// Mitsubishi GX Works2 project: plc0807   PLC: Q03UDV

PROGRAM MAIN
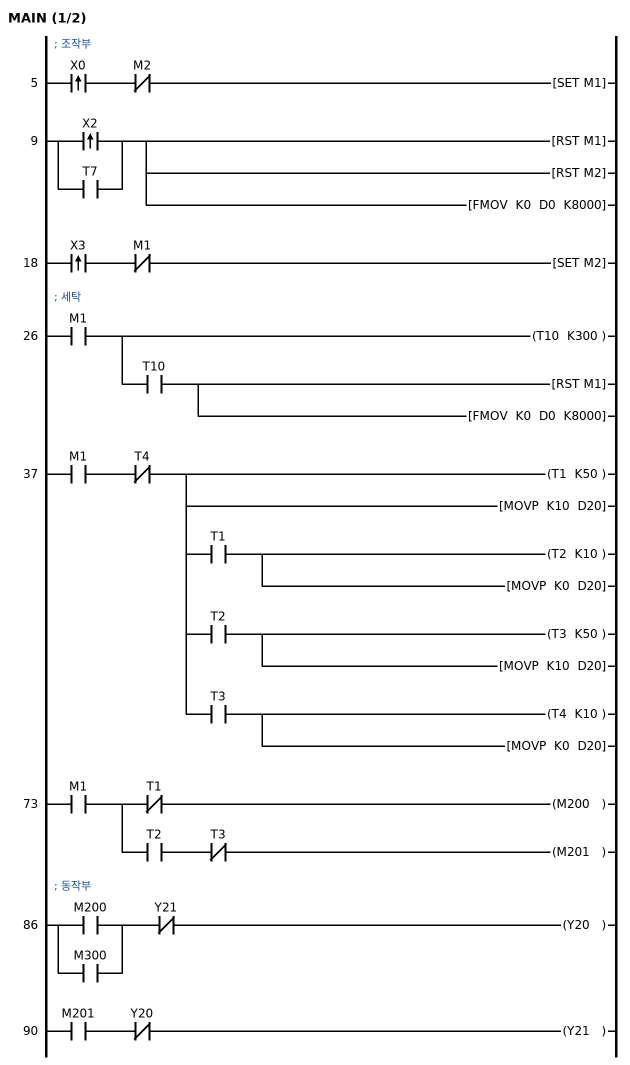
; 조작부
5     LDP     X0
      ANI     M2
      SET     M1
9     LDP     X2
      OR      T7
      RST     M1
      RST     M2
      FMOV    K0 D0 K8000
18    LDP     X3
      ANI     M1
      SET     M2
; 세탁
26    LD      M1
      OUT     T10 K300
      AND     T10
      RST     M1
      FMOV    K0 D0 K8000
37    LD      M1
      ANI     T4
      OUT     T1 K50
      MOVP    K10 D20
      MPS
      AND     T1
      OUT     T2 K10
      MOVP    K0 D20
      MRD
      AND     T2
      OUT     T3 K50
      MOVP    K10 D20
      MPP
      AND     T3
      OUT     T4 K10
      MOVP    K0 D20
73    LD      M1
      MPS
      ANI     T1
      OUT     M200
      MPP
      AND     T2
      ANI     T3
      OUT     M201
; 동작부
86    LD      M200
      OR      M300
      ANI     Y21
      OUT     Y20
90    LD      M201
      ANI     Y20
      OUT     Y21
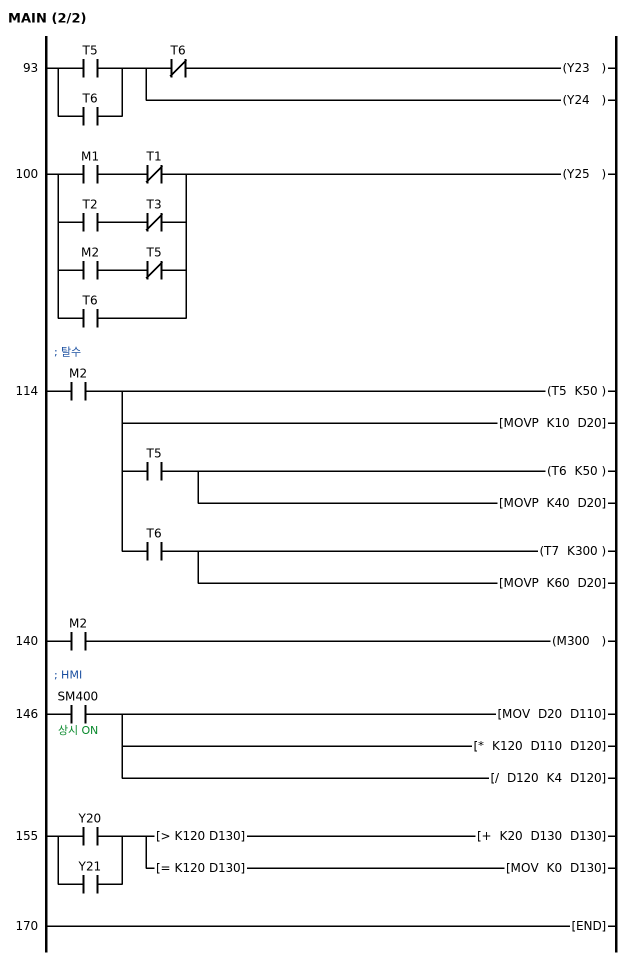
93    LD      T5
      OR      T6
      MPS
      ANI     T6
      OUT     Y23
      MPP
      OUT     Y24
100   LD      M1
      ANI     T1
      LD      T2
      ANI     T3
      ORB
      LD      M2
      ANI     T5
      ORB
      OR      T6
      OUT     Y25
; 탈수
114   LD      M2
      OUT     T5 K50
      MOVP    K10 D20
      MPS
      AND     T5
      OUT     T6 K50
      MOVP    K40 D20
      MPP
      AND     T6
      OUT     T7 K300
      MOVP    K60 D20
140   LD      M2
      OUT     M300
; HMI
146   LD      SM400  ; 상시 ON
      MOV     D20 D110
      *       K120 D110 D120
      /       D120 K4 D120
155   LD      Y20
      OR      Y21
      MPS
      AND>    K120 D130
      +       K20 D130 D130
      MPP
      AND=    K120 D130
      MOV     K0 D130
170   END
END_PROGRAM

PROGRAM inv15
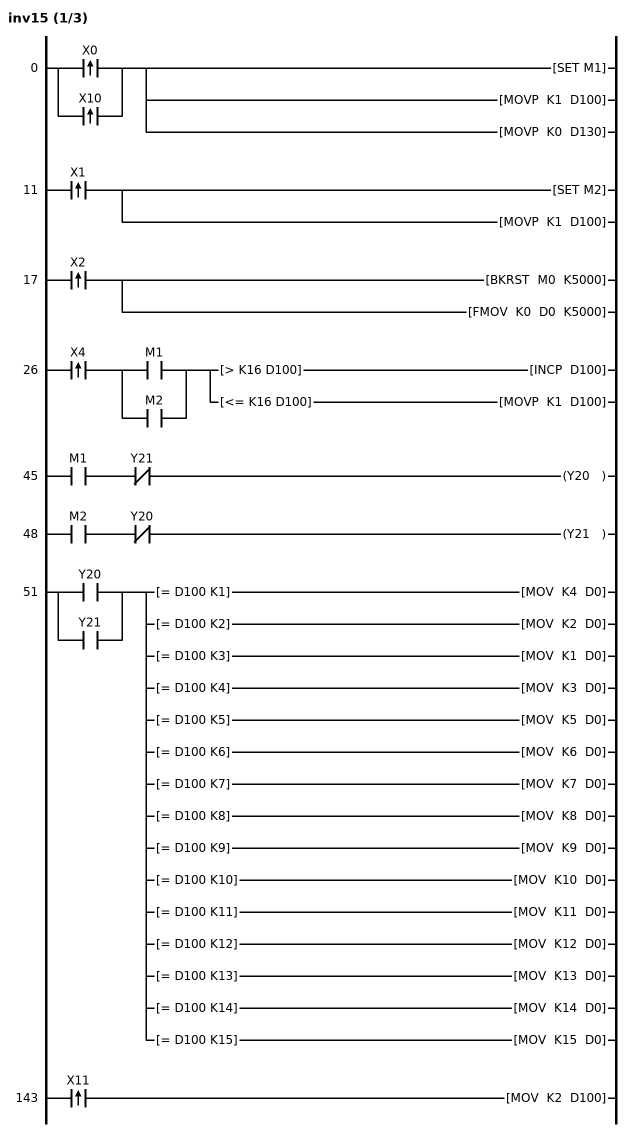
0     LDP     X0
      ORP     X10
      SET     M1
      MOVP    K1 D100
      MOVP    K0 D130
11    LDP     X1
      SET     M2
      MOVP    K1 D100
17    LDP     X2
      BKRST   M0 K5000
      FMOV    K0 D0 K5000
26    LDP     X4
      LD      M1
      OR      M2
      ANB
      MPS
      AND>    K16 D100
      INCP    D100
      MPP
      AND<=   K16 D100
      MOVP    K1 D100
45    LD      M1
      ANI     Y21
      OUT     Y20
48    LD      M2
      ANI     Y20
      OUT     Y21
51    LD      Y20
      OR      Y21
      MPS
      AND=    D100 K1
      MOV     K4 D0
      MRD
      AND=    D100 K2
      MOV     K2 D0
      MRD
      AND=    D100 K3
      MOV     K1 D0
      MRD
      AND=    D100 K4
      MOV     K3 D0
      MRD
      AND=    D100 K5
      MOV     K5 D0
      MRD
      AND=    D100 K6
      MOV     K6 D0
      MRD
      AND=    D100 K7
      MOV     K7 D0
      MRD
      AND=    D100 K8
      MOV     K8 D0
      MRD
      AND=    D100 K9
      MOV     K9 D0
      MRD
      AND=    D100 K10
      MOV     K10 D0
      MRD
      AND=    D100 K11
      MOV     K11 D0
      MRD
      AND=    D100 K12
      MOV     K12 D0
      MRD
      AND=    D100 K13
      MOV     K13 D0
      MRD
      AND=    D100 K14
      MOV     K14 D0
      MPP
      AND=    D100 K15
      MOV     K15 D0
143   LDP     X11
      MOV     K2 D100
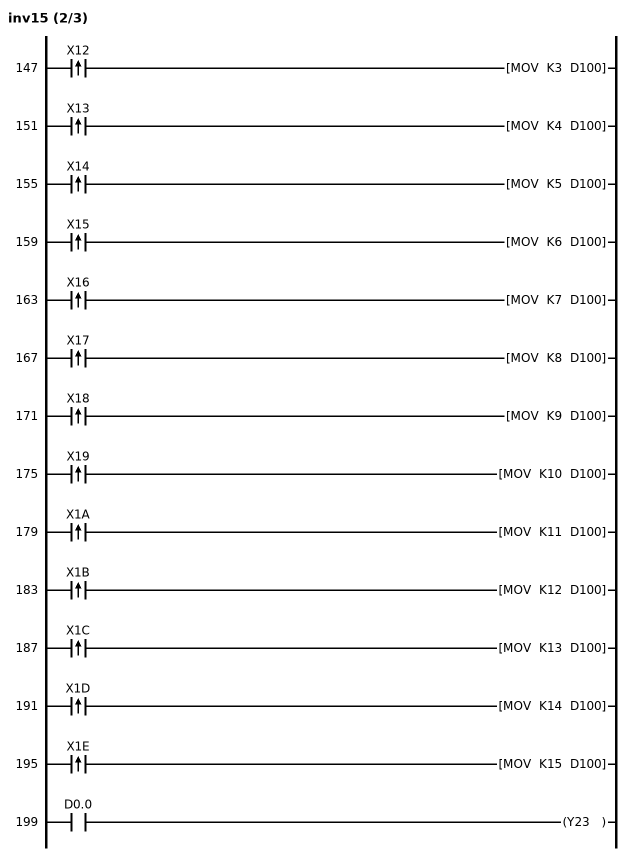
147   LDP     X12
      MOV     K3 D100
151   LDP     X13
      MOV     K4 D100
155   LDP     X14
      MOV     K5 D100
159   LDP     X15
      MOV     K6 D100
163   LDP     X16
      MOV     K7 D100
167   LDP     X17
      MOV     K8 D100
171   LDP     X18
      MOV     K9 D100
175   LDP     X19
      MOV     K10 D100
179   LDP     X1A
      MOV     K11 D100
183   LDP     X1B
      MOV     K12 D100
187   LDP     X1C
      MOV     K13 D100
191   LDP     X1D
      MOV     K14 D100
195   LDP     X1E
      MOV     K15 D100
199   LD      D0.0
      OUT     Y23
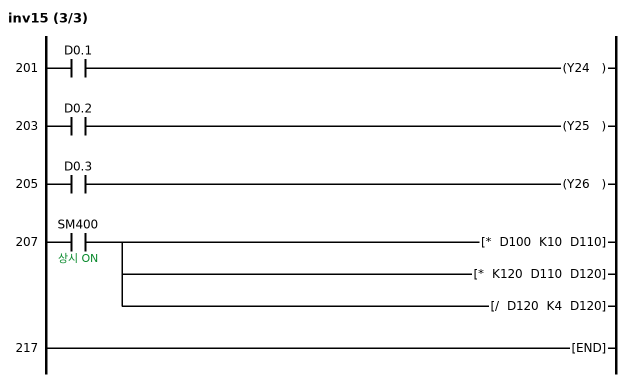
201   LD      D0.1
      OUT     Y24
203   LD      D0.2
      OUT     Y25
205   LD      D0.3
      OUT     Y26
207   LD      SM400  ; 상시 ON
      *       D100 K10 D110
      *       K120 D110 D120
      /       D120 K4 D120
217   END
END_PROGRAM

PROGRAM invDan
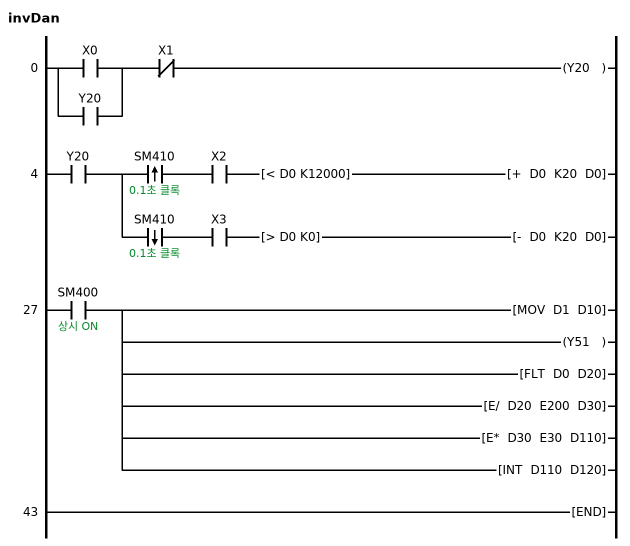
0     LD      X0
      OR      Y20
      ANI     X1
      OUT     Y20
4     LD      Y20
      MPS
      ANDP    SM410  ; 0.1초 클록
      AND     X2
      AND<    D0 K12000
      +       D0 K20 D0
      MPP
      ANDF    SM410  ; 0.1초 클록
      AND     X3
      AND>    D0 K0
      -       D0 K20 D0
27    LD      SM400  ; 상시 ON
      MOV     D1 D10
      OUT     Y51
      FLT     D0 D20
      E/      D20 E200 D30
      E*      D30 E30 D110
      INT     D110 D120
43    END
END_PROGRAM

PROGRAM Resist
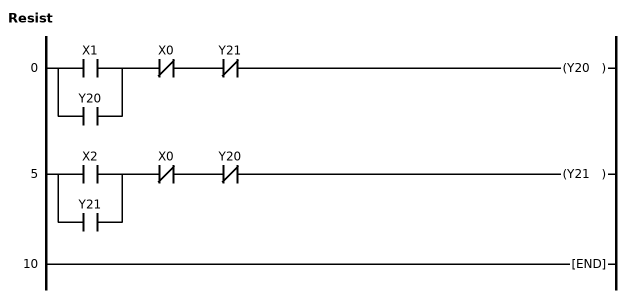
0     LD      X1
      OR      Y20
      ANI     X0
      ANI     Y21
      OUT     Y20
5     LD      X2
      OR      Y21
      ANI     X0
      ANI     Y20
      OUT     Y21
10    END
END_PROGRAM
